FUNCTION_BLOCK FB_MM710_IMU (* Service interface function block for Bosch MM7.10 IMU sensor via CAN/J1939 *)
  (* Standard: 61499-2; Description: Copyright (c) 2026 Meisterschulen am Ostbahnhof This program and the accompanying materials are made available under the terms of the Eclipse Public License 2.0 which is available at https://www.eclipse.org/legal/epl-2.0/ SPDX-License-Identifier: EPL-2.0 *)
  (* Version 1.0, 2026-04-24, AI, Meisterschulen am Ostbahnhof, Initial SIFB for MM710 IMU *)
  PACKAGE logiBUS::bosch::imu;
  IMPORT isobus::pgn::ISO_CAN_NODE;
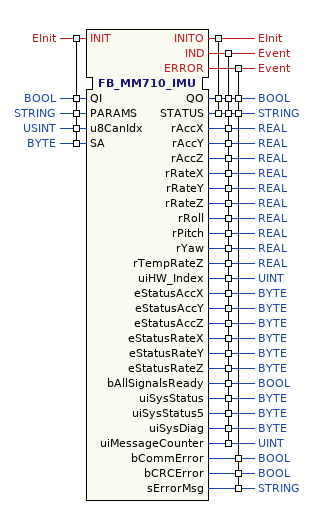
  EVENT_INPUT
    INIT : EInit WITH QI, PARAMS, u8CanIdx, SA; (* Service Initialization *)
  END_EVENT
  EVENT_OUTPUT
    INITO : EInit WITH QO, STATUS; (* Initialization Confirm *)
    IND WITH QO, STATUS, rAccX, rAccY, rAccZ, rRateX, rRateY, rRateZ, rRoll, rPitch, rYaw, rTempRateZ, uiHW_Index, eStatusAccX, eStatusAccY, eStatusAccZ, eStatusRateX, eStatusRateY, eStatusRateZ, bAllSignalsReady, uiSysStatus, uiSysStatus5, uiSysDiag, uiMessageCounter; (* Indication from Resource *)
    ERROR WITH QO, STATUS, bCommError, bCRCError, sErrorMsg; (* Error indication *)
  END_EVENT
  VAR_INPUT
    QI : BOOL; (* Event Input Qualifier *)
    PARAMS : STRING; (* Service Parameters (e.g. CAN interface config) *)
    u8CanIdx : USINT := ISO_CAN_NODE::INVALID; (* ISO_CAN_NODE *)
    SA : BYTE := 16#DA; (* Source Address *)
  END_VAR
  VAR_OUTPUT
    QO : BOOL; (* Event Output Qualifier *)
    STATUS : STRING; (* Service Status *)
    rAccX : REAL; (* Acceleration X [m/s^2] *)
    rAccY : REAL; (* Acceleration Y [m/s^2] *)
    rAccZ : REAL; (* Acceleration Z [m/s^2] *)
    rRateX : REAL; (* Rotation rate X [deg/s] *)
    rRateY : REAL; (* Rotation rate Y [deg/s] *)
    rRateZ : REAL; (* Rotation rate Z [deg/s] *)
    rRoll : REAL; (* Inclination Roll [deg] *)
    rPitch : REAL; (* Inclination Pitch [deg] *)
    rYaw : REAL; (* Inclination Yaw [deg] *)
    rTempRateZ : REAL; (* Sensor temperature [degC] *)
    uiHW_Index : UINT; (* Hardware index (0=MM5.10, 1=MM7.10) *)
    eStatusAccX : BYTE; (* Signal status AccX (0=ready, 1..7=error) *)
    eStatusAccY : BYTE; (* Signal status AccY (0=ready, 1..7=error) *)
    eStatusAccZ : BYTE; (* Signal status AccZ (0=ready, 1..7=error) *)
    eStatusRateX : BYTE; (* Signal status RateX (0=ready, 1..7=error) *)
    eStatusRateY : BYTE; (* Signal status RateY (0=ready, 1..7=error) *)
    eStatusRateZ : BYTE; (* Signal status RateZ (0=ready, 1..7=error) *)
    bAllSignalsReady : BOOL; (* TRUE if all status = 0 *)
    uiSysStatus : BYTE; (* System status (from TX1) *)
    uiSysStatus5 : BYTE; (* System status (from TX2) *)
    uiSysDiag : BYTE; (* System diagnostic code (from TX2) *)
    uiMessageCounter : UINT; (* Message counter (0..15) for timeout monitoring *)
    bCommError : BOOL; (* TRUE if CAN timeout exceeded *)
    bCRCError : BOOL; (* TRUE if CRC check failed *)
    sErrorMsg : STRING; (* Error message text *)
  END_VAR
END_FUNCTION_BLOCK
